# EPICS autosave request: FOFBApp/Db/FOFBTrigger_settings.req
$(P)$(R)$(TRIGGER_NAME)$(TRIGGER_CHAN)Dir-Sel
$(P)$(R)$(TRIGGER_NAME)$(TRIGGER_CHAN)DirPol-Sel
$(P)$(R)$(TRIGGER_NAME)$(TRIGGER_CHAN)RcvLen-SP
$(P)$(R)$(TRIGGER_NAME)$(TRIGGER_CHAN)TrnLen-SP
$(P)$(R)$(TRIGGER_NAME)$(TRIGGER_CHAN)RcvSrc-Sel
$(P)$(R)$(TRIGGER_NAME)$(TRIGGER_CHAN)TrnSrc-Sel
$(P)$(R)$(TRIGGER_NAME)$(TRIGGER_CHAN)RcvInSel-SP
$(P)$(R)$(TRIGGER_NAME)$(TRIGGER_CHAN)TrnOutSel-SP
